PROGRAM ShortProcess
VAR
	cM1startCount : INT;
	
END_VAR
// written 7.08.2023 by Daniel Kelly

// Program is a shorter version of the full process cycle

//Step RValveOff turns off the top and bottom closing valves
// Step Wait500 waits until the temperature is at 500
//Step GasFanOn turns on the gas fan
// Step waittemp is the residence time
//Step ShortFeed and Biomass Feed run simultaneously to feed the biomass into the furnace
// Step ExitMotor operates the removal motor and opens the top valve
// Steps M1override and M2override overrides the original motor operating time.
//Step Valve2Open opens the bottom valve
// Step Valve2Close closes the bottom valve

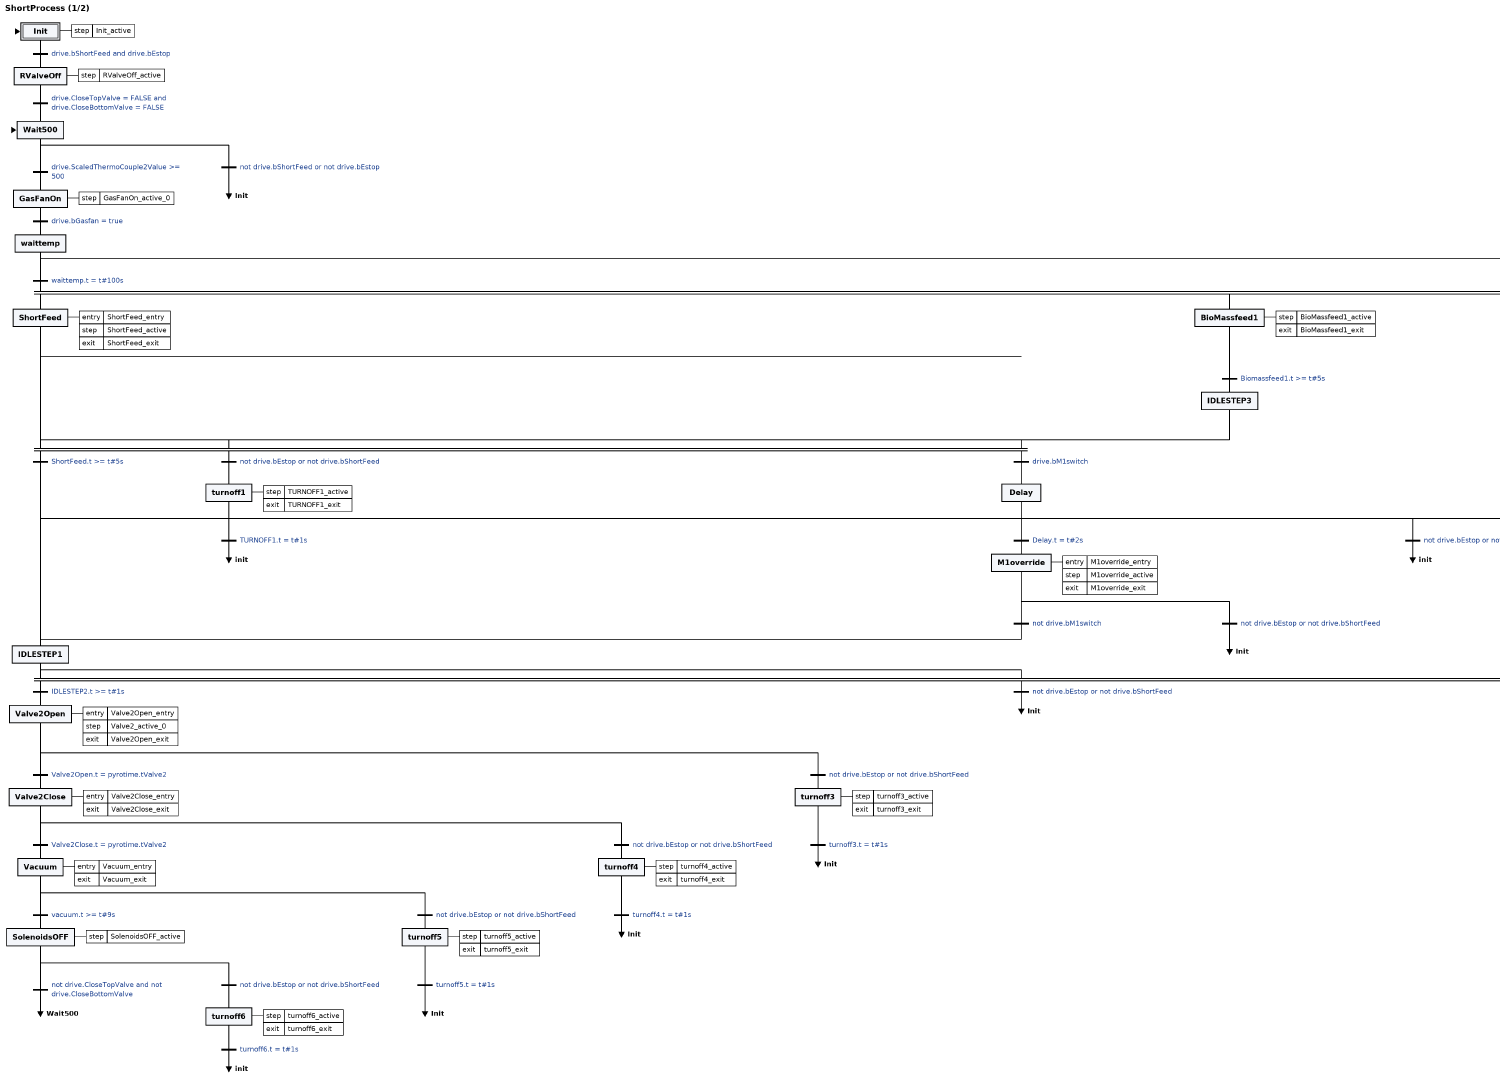
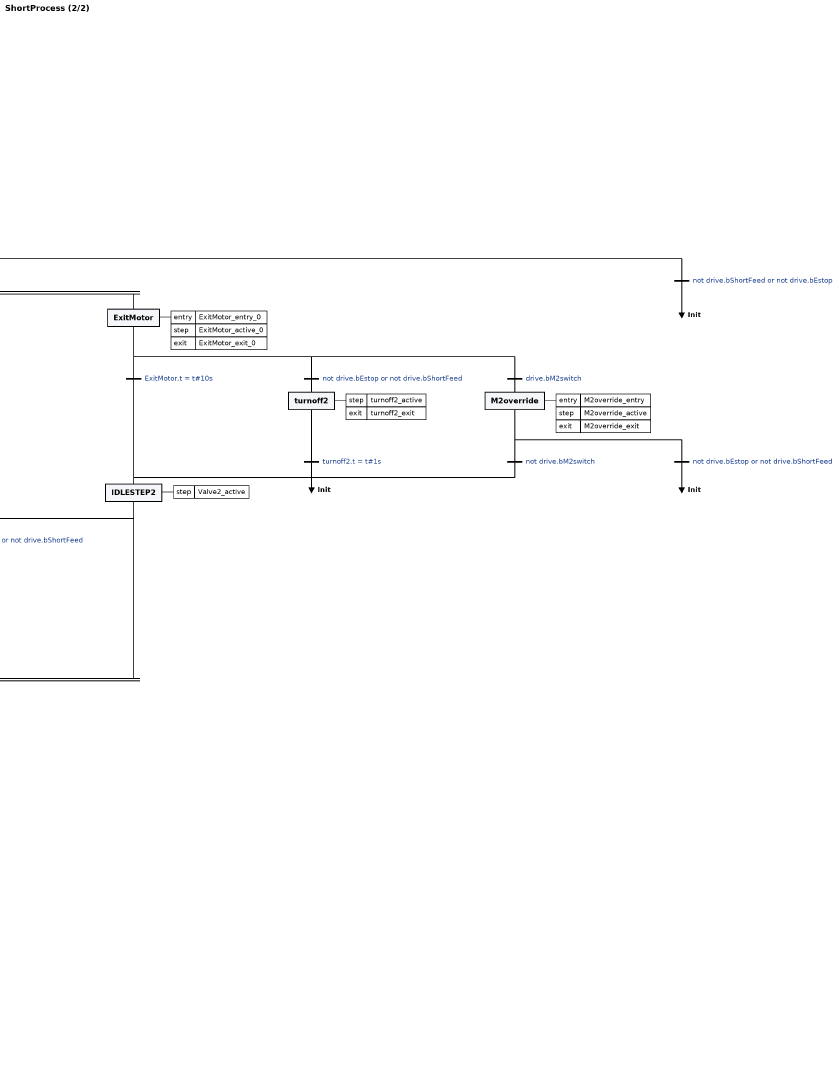
INITIAL_STEP Init:
    Init_active(N);  // step action
END_STEP
TRANSITION FROM Init TO RValveOff
    := drive.bShortFeed and drive.bEstop;
END_TRANSITION
STEP RValveOff:
    RValveOff_active(N);  // step action
END_STEP
TRANSITION FROM RValveOff TO Wait500
    := drive.CloseTopValve = FALSE and drive.CloseBottomValve = FALSE;
END_TRANSITION
STEP Wait500:
END_STEP
TRANSITION FROM Wait500 TO GasFanOn
    := drive.ScaledThermoCouple2Value >= 500;
END_TRANSITION
STEP GasFanOn:
    GasFanOn_active_0(N);  // step action
END_STEP
TRANSITION FROM GasFanOn TO waittemp
    := drive.bGasfan = true;
END_TRANSITION
TRANSITION FROM Wait500 TO Init
    := not drive.bShortFeed or not drive.bEstop;
END_TRANSITION
STEP waittemp:
END_STEP
TRANSITION FROM waittemp TO (ShortFeed, BioMassfeed1, ExitMotor)
    := waittemp.t = t#100s;
END_TRANSITION
TRANSITION FROM waittemp TO Init
    := not drive.bShortFeed or not drive.bEstop;
END_TRANSITION
STEP ShortFeed:
    ShortFeed_entry(P1);  // entry action
    ShortFeed_active(N);  // step action
    ShortFeed_exit(P0);  // exit action
END_STEP
STEP BioMassfeed1:
    BioMassfeed1_active(N);  // step action
    BioMassfeed1_exit(P0);  // exit action
END_STEP
TRANSITION FROM BioMassfeed1 TO IDLESTEP3
    := Biomassfeed1.t >= t#5s;
END_TRANSITION
STEP IDLESTEP3:
END_STEP
TRANSITION FROM (ShortFeed, IDLESTEP3) TO IDLESTEP1
    := ShortFeed.t >= t#5s;
END_TRANSITION
TRANSITION FROM (ShortFeed, IDLESTEP3) TO turnoff1
    := not drive.bEstop or not drive.bShortFeed;
END_TRANSITION
STEP turnoff1:
    TURNOFF1_active(N);  // step action
    TURNOFF1_exit(P0);  // exit action
END_STEP
TRANSITION FROM turnoff1 TO init
    := TURNOFF1.t = t#1s;
END_TRANSITION
TRANSITION FROM (ShortFeed, IDLESTEP3) TO Delay
    := drive.bM1switch;
END_TRANSITION
STEP Delay:
END_STEP
TRANSITION FROM Delay TO M1override
    := Delay.t = t#2s;
END_TRANSITION
TRANSITION FROM Delay TO init
    := not drive.bEstop or not drive.bShortFeed;
END_TRANSITION
STEP M1override:
    M1override_entry(P1);  // entry action
    M1override_active(N);  // step action
    M1override_exit(P0);  // exit action
END_STEP
TRANSITION FROM M1override TO IDLESTEP1
    := not drive.bM1switch;
END_TRANSITION
TRANSITION FROM M1override TO Init
    := not drive.bEstop or not drive.bShortFeed;
END_TRANSITION
STEP IDLESTEP1:
END_STEP
STEP ExitMotor:
    ExitMotor_entry_0(P1);  // entry action
    ExitMotor_active_0(N);  // step action
    ExitMotor_exit_0(P0);  // exit action
END_STEP
TRANSITION FROM ExitMotor TO IDLESTEP2
    := ExitMotor.t = t#10s;
END_TRANSITION
TRANSITION FROM ExitMotor TO turnoff2
    := not drive.bEstop or not drive.bShortFeed;
END_TRANSITION
STEP turnoff2:
    turnoff2_active(N);  // step action
    turnoff2_exit(P0);  // exit action
END_STEP
TRANSITION FROM turnoff2 TO Init
    := turnoff2.t = t#1s;
END_TRANSITION
TRANSITION FROM ExitMotor TO M2override
    := drive.bM2switch;
END_TRANSITION
STEP M2override:
    M2override_entry(P1);  // entry action
    M2override_active(N);  // step action
    M2override_exit(P0);  // exit action
END_STEP
TRANSITION FROM M2override TO IDLESTEP2
    := not drive.bM2switch;
END_TRANSITION
TRANSITION FROM M2override TO Init
    := not drive.bEstop or not drive.bShortFeed;
END_TRANSITION
STEP IDLESTEP2:
    Valve2_active(N);  // step action
END_STEP
TRANSITION FROM (IDLESTEP1, IDLESTEP2) TO Valve2Open
    := IDLESTEP2.t >= t#1s;
END_TRANSITION
TRANSITION FROM (IDLESTEP1, IDLESTEP2) TO Init
    := not drive.bEstop or not drive.bShortFeed;
END_TRANSITION
STEP Valve2Open:
    Valve2Open_entry(P1);  // entry action
    Valve2_active_0(N);  // step action
    Valve2Open_exit(P0);  // exit action
END_STEP
TRANSITION FROM Valve2Open TO Valve2Close
    := Valve2Open.t = pyrotime.tValve2;
END_TRANSITION
TRANSITION FROM Valve2Open TO turnoff3
    := not drive.bEstop or not drive.bShortFeed;
END_TRANSITION
STEP turnoff3:
    turnoff3_active(N);  // step action
    turnoff3_exit(P0);  // exit action
END_STEP
TRANSITION FROM turnoff3 TO Init
    := turnoff3.t = t#1s;
END_TRANSITION
STEP Valve2Close:
    Valve2Close_entry(P1);  // entry action
    Valve2Close_exit(P0);  // exit action
END_STEP
TRANSITION FROM Valve2Close TO Vacuum
    := Valve2Close.t = pyrotime.tValve2;
END_TRANSITION
TRANSITION FROM Valve2Close TO turnoff4
    := not drive.bEstop or not drive.bShortFeed;
END_TRANSITION
STEP turnoff4:
    turnoff4_active(N);  // step action
    turnoff4_exit(P0);  // exit action
END_STEP
TRANSITION FROM turnoff4 TO Init
    := turnoff4.t = t#1s;
END_TRANSITION
STEP Vacuum:
    Vacuum_entry(P1);  // entry action
    Vacuum_exit(P0);  // exit action
END_STEP
TRANSITION FROM Vacuum TO SolenoidsOFF
    := vacuum.t >= t#9s;
END_TRANSITION
TRANSITION FROM Vacuum TO turnoff5
    := not drive.bEstop or not drive.bShortFeed;
END_TRANSITION
STEP turnoff5:
    turnoff5_active(N);  // step action
    turnoff5_exit(P0);  // exit action
END_STEP
TRANSITION FROM turnoff5 TO Init
    := turnoff5.t = t#1s;
END_TRANSITION
STEP SolenoidsOFF:
    SolenoidsOFF_active(N);  // step action
END_STEP
TRANSITION FROM SolenoidsOFF TO Wait500
    := not drive.CloseTopValve and not drive.CloseBottomValve;
END_TRANSITION
TRANSITION FROM SolenoidsOFF TO turnoff6
    := not drive.bEstop or not drive.bShortFeed;
END_TRANSITION
STEP turnoff6:
    turnoff6_active(N);  // step action
    turnoff6_exit(P0);  // exit action
END_STEP
TRANSITION FROM turnoff6 TO init
    := turnoff6.t = t#1s;
END_TRANSITION

ACTION BioMassfeed1_active:
drive.bFeedMotor2 := TRUE;
drive.bFeedMotor2Lamp := TRUE;
END_ACTION

ACTION BioMassfeed1_exit:
drive.bFeedMotor2 := FALSE;
drive.bFeedMotor2Lamp := FALSE;
END_ACTION

ACTION ExitMotor_active_0:
drive.bRemovalMotor := TRUE; 
drive.bM2active := TRUE; // turns on the lamp

drive.bValveLamp := TRUE; // turns on the valve lamp
drive.OpenTopValve := TRUE; 
drive.CloseTopValve := FALSE;
END_ACTION

ACTION ExitMotor_entry_0:

END_ACTION

ACTION ExitMotor_exit_0:

IF drive.OpenTopValve THEN 
	drive.itopvalvecount := drive.itopvalvecount + 1;
END_IF



drive.CloseTopValve := TRUE;
drive.OpenTopValve := FALSE;



drive.bM2active := FALSE; // lamp off
drive.bRemovalMotor := FALSE;
END_ACTION

ACTION ExitMotor1_active:
drive.bRemovalMotor := TRUE;
END_ACTION

ACTION GasFanOFF_active:
drive.bGasfan := FALSE;
END_ACTION

ACTION GasFanOn_active:
drive.bGasfan := true;
END_ACTION

ACTION GasFanOn_active_0:
drive.bGasfan := true;
END_ACTION

ACTION Init_active:
//drive.ATV_RPDO_Output1_Control_Word := 0;
//drive.bRemovalMotor := FALSE;
//drive.bProcessActive := FALSE; 
//drive.LeftSolenoid := FALSE;
//drive.LeftSolenoid2 := FALSE; 
//drive.RightSolenoid := TRUE;
//drive.RightSolenoid2 := TRUE;

drive.bGasfan := FALSE;
END_ACTION

ACTION Init_Feeding_active:
IF drive.ATV_TPDO_Input1_Status_Word = ATV_Status.rdy2SwitchON THEN 
	drive.ATV_RPDO_Output1_Control_Word := 7; //SwitchedON
END_IF

IF drive.ATV_TPDO_Input1_Status_Word = ATV_Status.SwitchedON THEN 
	drive.ATV_RPDO_Output1_Control_Word := 15; //OP_Enabled
END_IF
END_ACTION

ACTION Init_Feeding_entry:
drive.ATV_RPDO_Output1_Control_Word := 6; //rdy2SwitchON
drive.ATV_RPDO_Output2_Target_Velocity := 1000;
END_ACTION

ACTION Init_Feeding_exit:
drive.ATV_RPDO_Output1_Control_Word := 7; //switchedON
END_ACTION

ACTION M1override_active:
IF drive.ATV_TPDO_Input1_Status_Word = atv_status.rdy2SwitchON THEN 
	drive.ATV_RPDO_Output1_Control_Word := 7;
END_IF

IF drive.ATV_TPDO_Input1_Status_Word = atv_status.SwitchedON THEN 
	drive.ATV_RPDO_Output1_Control_Word := 15;
	drive.bM1active := TRUE; 
END_IF
END_ACTION

ACTION M1override_entry:
drive.ATV_RPDO_Output2_Target_Velocity := 1000;
drive.ATV_RPDO_Output1_Control_Word := 6;
END_ACTION

ACTION M1override_exit:
drive.ATV_RPDO_Output1_Control_Word := 7; 
drive.bM1active := false;
END_ACTION

ACTION M2override_active:

END_ACTION

ACTION M2override_entry:
drive.bRemovalMotor := TRUE; 
drive.bM2active := TRUE;
END_ACTION

ACTION M2override_exit:
drive.bRemovalMotor := FALSE; 
drive.bM2active := FALSE;
END_ACTION

ACTION ProcessACTIVE_active:
drive.bProcessActive := TRUE;
END_ACTION

ACTION RValveOff_active:
drive.CloseTopValve := FALSE;
drive.CloseBottomValve := FALSE;
END_ACTION

ACTION ShortFeed_active:
drive.bRemovalMotor := TRUE;
drive.bM1active := TRUE;

IF drive.ATV_TPDO_Input1_Status_Word = ATV_Status.rdy2SwitchON THEN 
	drive.ATV_RPDO_Output1_Control_Word := 7;
END_IF

IF drive.ATV_TPDO_Input1_Status_Word = ATV_Status.SwitchedON THEN
			drive.bM1run := TRUE; 
			drive.ATV_RPDO_Output1_Control_Word := 15;
END_IF
END_ACTION

ACTION ShortFeed_entry:
drive.ATV_RPDO_Output2_Target_Velocity := 1000;
drive.ATV_RPDO_Output1_Control_Word := 6;
END_ACTION

ACTION ShortFeed_exit:
IF drive.bM1run = TRUE THEN 
	cM1startCount := cM1startCount + 1;
END_IF

drive.bM1run := FALSE;
drive.bM1active := FALSE; 
drive.ATV_RPDO_Output1_Control_Word := 7;
END_ACTION

ACTION SolenoidsOFF_active:
drive.CloseTopValve := FALSE;
drive.CloseBottomValve := FALSE;
END_ACTION

ACTION TURNOFF1_active:
drive.bRemovalMotor := FALSE;
drive.OpenTopValve := FALSE;
drive.CloseTopValve := TRUE;
drive.bM1active := false;
END_ACTION

ACTION TURNOFF1_exit:
drive.CloseBottomValve := FALSE;
drive.CloseTopValve := FALSE;
END_ACTION

ACTION turnoff2_active:
drive.bRemovalMotor := FALSE;
drive.OpenTopValve := FALSE;
drive.CloseTopValve := TRUE;
END_ACTION

ACTION turnoff2_exit:
drive.CloseBottomValve := FALSE;
drive.CloseTopValve := FALSE;
END_ACTION

ACTION turnoff3_active:
drive.bRemovalMotor := FALSE;
drive.OpenTopValve := FALSE;
drive.CloseTopValve := TRUE;
drive.OpenBottomValve := FALSE;
drive.CloseBottomValve := TRUE;
END_ACTION

ACTION turnoff3_exit:
drive.CloseBottomValve := FALSE;
drive.CloseTopValve := FALSE;
END_ACTION

ACTION turnoff4_active:
drive.bRemovalMotor := FALSE;
drive.OpenTopValve := FALSE;
drive.CloseTopValve := TRUE;
drive.OpenBottomValve := FALSE;
drive.CloseBottomValve := TRUE;
END_ACTION

ACTION turnoff4_exit:
drive.CloseBottomValve := FALSE;
drive.CloseTopValve := FALSE;
END_ACTION

ACTION turnoff5_active:
drive.bRemovalMotor := FALSE;
drive.OpenTopValve := FALSE;
drive.CloseTopValve := TRUE;
drive.OpenBottomValve := FALSE;
drive.CloseBottomValve := TRUE;
END_ACTION

ACTION turnoff5_exit:
drive.CloseBottomValve := FALSE;
drive.CloseTopValve := FALSE;
END_ACTION

ACTION turnoff6_active:
drive.bRemovalMotor := FALSE;
drive.OpenTopValve := FALSE;
drive.CloseTopValve := TRUE;
drive.OpenBottomValve := FALSE;
drive.CloseBottomValve := TRUE;
END_ACTION

ACTION turnoff6_exit:
drive.CloseBottomValve := FALSE;
drive.CloseTopValve := FALSE;
END_ACTION

ACTION Vacuum_entry:
IF drive.itopvalvecount >= 5 THEN 
	drive.bVacuum := TRUE; 
END_IF
END_ACTION

ACTION Vacuum_exit:
drive.bVacuum := FALSE;
END_ACTION

ACTION Valve2_active:

END_ACTION

ACTION Valve2_active_0:

END_ACTION

ACTION Valve2_exit:

END_ACTION

ACTION Valve2Close_entry:
drive.CloseBottomValve := TRUE;
END_ACTION

ACTION Valve2Close_exit:
drive.CloseBottomValve := FALSE;
drive.bValveLamp := FALSE;
END_ACTION

ACTION Valve2Open_entry:

IF drive.itopvalvecount >= 5 THEN // Bottom valve opens after top valve has opened 5 times or more
	drive.OpenBottomValve := TRUE;
END_IF
END_ACTION

ACTION Valve2Open_exit:

IF drive.OpenBottomValve THEN  //  counter will reset after bottom valve opens
	drive.itopvalvecount := 1; 
END_IF

drive.OpenBottomValve := FALSE;
END_ACTION

END_PROGRAM

(* stored: Version 1.1.0.1, ProductVersion 3.1.4024.12
   POU ShortProcess: Id {6eb4231c-84a3-4f52-91bb-a80605e07848}, SpecialFunc None
   Folder VISUs: Id {daf3baf7-37f1-4e01-9da9-70c42a5204c2}
   Action BioMassfeed1_active: Id {7fa01ed5-4a23-4c43-9663-ddff64d49b88}
   Action BioMassfeed1_exit: Id {8ff846c4-f66b-4cca-9c7c-c0424a40d4fe}
   Action ExitMotor_active_0: Id {9e241222-ec61-4a48-aed7-629e2eb21d49}
   Action ExitMotor_entry_0: Id {e6bb01f5-1372-49cc-bdae-216ff50231fd}
   Action ExitMotor_exit_0: Id {651105aa-a2c8-4ee3-b7e1-70e730f81695}
   Action ExitMotor1_active: Id {6eb9fd99-a635-477a-a929-e60232b5725b}
   Action GasFanOFF_active: Id {470acc8a-e483-49e3-b192-9e65ae945e73}
   Action GasFanOn_active: Id {a053e862-164f-4d0d-8bee-fe2e0e05ffe1}
   Action GasFanOn_active_0: Id {0b0b785e-af64-437a-8cb1-3424963e42e2}
   Action Init_active: Id {c1ed9047-b84e-429f-8b92-b7dfbc514801}
   Action Init_Feeding_active: Id {391a720e-ef48-45ef-8cc5-63c70b8481dd}
   Action Init_Feeding_entry: Id {06e85772-aacf-437f-9bad-ca28ec5e6b79}
   Action Init_Feeding_exit: Id {d5b21758-ed34-4946-b9b4-69b1c6a1601f}
   Action M1override_active: Id {bd4b9e56-e762-4a54-88ab-5c0820e9afd8}
   Action M1override_entry: Id {0e9f096a-5ead-4b7b-af3e-0c2095114c55}
   Action M1override_exit: Id {58f7992f-a7a8-4a90-94e0-64b55bdc9c1a}
   Action M2override_active: Id {e24662cb-df54-49e7-96e3-ed2458ef3fa0}
   Action M2override_entry: Id {e50194a6-a93e-4fce-a44d-b4acd5932eab}
   Action M2override_exit: Id {debeb8f5-c6d9-4350-b67c-5434e9e69890}
   Action ProcessACTIVE_active: Id {c6181bf7-3139-485d-8f53-982e972e9b42}
   Action RValveOff_active: Id {adf1ceb9-7cba-43da-b347-e66922cc2edb}
   Action ShortFeed_active: Id {3b0f0261-da2a-4594-97fc-3f1d7aa1ffee}
   Action ShortFeed_entry: Id {9100713d-f773-4970-ae58-77ab7bdc8e70}
   Action ShortFeed_exit: Id {4e905060-4eeb-4d50-919e-c024b0618e63}
   Action SolenoidsOFF_active: Id {7bc41ecd-27ca-4594-b9f1-aae51a28374f}
   Action TURNOFF1_active: Id {e0ddb214-3d89-42cb-b2f5-55dd30feff40}
   Action TURNOFF1_exit: Id {4a2c41e4-b424-42e2-85ba-7549623b4800}
   Action turnoff2_active: Id {2f1f01d2-3dc4-4c1d-bb54-40755f328ba7}
   Action turnoff2_exit: Id {19fc746f-0a75-4471-8ce3-461b65eb7e24}
   Action turnoff3_active: Id {d819df9b-0506-4cf2-a9fc-ccea3ee10b69}
   Action turnoff3_exit: Id {a86f4c55-734d-4871-a116-f7591e5a6980}
   Action turnoff4_active: Id {6fc7b9d8-c54d-464b-a521-fd653df5b089}
   Action turnoff4_exit: Id {00d7b4cf-064a-42cc-b42f-e4f07762c3fa}
   Action turnoff5_active: Id {3d42cf2e-bb10-4be5-a050-6ae33ae9b4af}
   Action turnoff5_exit: Id {27aba626-3787-4cc0-ae3d-f12bfc16c783}
   Action turnoff6_active: Id {7d8fc17d-6452-4b0e-9ee3-98cc86e8b48c}
   Action turnoff6_exit: Id {fa5bfbcd-2672-483c-9ea1-331f9dfde07e}
   Action Vacuum_entry: Id {d2373440-0776-481d-819b-3cabf1795ae8}
   Action Vacuum_exit: Id {6057b437-dd4d-41cf-a599-23aa22ab735c}
   Action Valve2_active: Id {5d308012-97b5-4d6e-b066-a7833da06817}
   Action Valve2_active_0: Id {7d578137-3f04-4862-a39f-e621de5210f7}
   Action Valve2_exit: Id {e9fad988-59d4-4010-a0c0-69b35344a8f4}
   Action Valve2Close_entry: Id {cb297ce2-569b-4895-849e-717227893205}
   Action Valve2Close_exit: Id {e4fce59f-e072-4665-995e-8d4c56fcd8d0}
   Action Valve2Open_entry: Id {36c4da84-89e3-49ac-8800-434b548a5dc7}
   Action Valve2Open_exit: Id {0ec6f428-d782-41e2-8def-a2573399d570} *)
